{attribute 'linkalways'} 
{attribute 'no_explicit_call' := 'This FB is a CLASS and must be accessed using methods or properties'}
{attribute 'enable_dynamic_creation'}
FUNCTION_BLOCK Node_F_VN_MinElementElementwise_LREAL EXTENDS VisionNode
VAR
    ipContainer : _ITcVnContainer;
    fMin : _LREAL(0.0);
    hrPrev : _HRESULT(S_OK);
    hresult : _HRESULT(S_OK);
END_VAR

METHOD PUBLIC  Clone : I_Node
VAR
	pNode : POINTER TO Node_F_VN_MinElementElementwise_LREAL;
END_VAR
pNode := __NEW(Node_F_VN_MinElementElementwise_LREAL);
Clone := pNode^;
END_METHOD

METHOD FB_init : BOOL
VAR_INPUT
	bInitRetains : BOOL; // if TRUE, the retain variables are initialized (warm start / cold start)
	bInCopyCode : BOOL;  // if TRUE, the instance afterwards gets moved into the copy code (online change)
END_VAR
AddInput('ipContainer', ipContainer);
AddInput('fMin', fMin);
AddInput('hrPrev', hrPrev);
AddOutput('ipContainer', ipContainer);
AddOutput('hresult',hresult);
END_METHOD

METHOD PROTECTED OnExecute : HRESULT
hresult.Value := F_VN_MinElementElementwise_LREAL(
    ipContainer := ipContainer.Value,
    fMin := fMin.Value,
    hrPrev:= hrPrev.Value);
END_METHOD

METHOD PUBLIC PreExecutionCheck
VAR_INPUT
	Check : I_PreExecutionChecks;
END_VAR
Check.IsTrue(ipContainer.IsValid, 'ipContainer must be a valid container');
Check.IsTrue(ipContainer.HasType('CTcVnContainer_Vector_LREAL'), 'ipContainer contains incorrect types');
END_METHOD

END_FUNCTION_BLOCK

(* stored: Version 1.1.0.1, ProductVersion 3.1.4024.13
   POU Node_F_VN_MinElementElementwise_LREAL: Id {7753e2ae-7d64-4d29-932a-297a0bab9637}, SpecialFunc None
   Folder Constructor: Id {b68b6ec5-6c44-4d01-bb62-f7d533e95b00}
   Method Clone: Id {1846edf2-ad0c-4bdf-b4b1-a2fc3ada2020}
   Method FB_init: Id {0726b24b-3af2-4511-b326-4c69e6e4abe1}
   Method OnExecute: Id {f52214ac-55f0-4bca-a475-79aa32a4d9a9}
   Method PreExecutionCheck: Id {23b96f82-5de2-471f-8101-71f3726eaf21} *)
